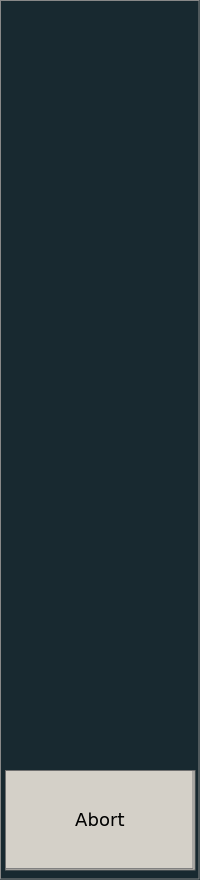
VISUALIZATION NavBarInitializing  // 200x880
VAR_IN_OUT
	btnAbort : BOOL;
END_VAR
    Button (5,770 190x100), "Abort"
        tap btnAbort
END_VISUALIZATION

(* stored: Version 1.1.0.1, ProductVersion 3.1.4024.9
   Visu NavBarInitializing: Id {dfc84bfc-40f9-4679-ba57-0e8c0dc01e68} *)
